TYPE TcoUrRoboticsOutputData : STRUCT
    {attribute addProperty Name "<#Speed#>"}
    Speed : TcoUrRobotics_O2TRobot;
    {attribute addProperty Name "<#IO#>"}
    IO : TcoUrRobotics_O2TIo;
    {attribute addProperty Name "<#Reg 1#>"}
    Reg1 : TcoUrRobotics_O2TReg;
    {attribute addProperty Name "<#Reg 2#>"}
    Reg2 : TcoUrRobotics_O2TReg;
END_STRUCT
END_TYPE

(* stored: Version 1.1.0.1, ProductVersion 3.1.4024.12
   DUT TcoUrRoboticsOutputData: Id {0f2afbca-1c3f-0669-1377-25c97b69294d} *)
